{attribute 'qualified_only'}
VAR_GLOBAL CONSTANT
END_VAR

(* stored: Version 1.1.0.1, ProductVersion 3.1.4024.11
   GVL Param: Id {d99940d7-24b9-429b-bbb4-17292851c71f}, ParameterList True *)
